FUNCTION_BLOCK FB_StepperHoming EXTENDS FB_StateMachine IMPLEMENTS  I_StateMachine
VAR_INPUT
	bStart : BOOL;	
	
	stParentsAxis : REFERENCE TO ST_StepperAxis;
	
END_VAR
VAR_OUTPUT
END_VAR
VAR
	eInnerState : E_StepperHomingStates;
	bCompleted : BOOL;
	dtTimeCompleted: DATE_AND_TIME;
	
	bEnabledBeforeHoming : BOOL;
	bOutsideHome AT %I* : BOOL;
	fRelativePosition 		: LREAL;
	fAbsolutePosition		: LREAL;
	
	stAxisRef : REFERENCE TO AXIS_REF;
	fbPower : MC_Power;
	fbReset :MC_Reset;
	fbHalt : MC_Halt;
	fbJog : MC_JOG;
	fbHome : MC_Home;
	bOutwardsForward	: REFERENCE TO BOOL;
	bOutwardsBackwards	: REFERENCE TO BOOL;
	bInwardsForward		: REFERENCE TO BOOL;
	bInwardsBackwards	: REFERENCE TO BOOL;
	fHomePosition		: REFERENCE TO LREAL;
	bForceHoming : REFERENCE TO BOOL;
	nPLC_Cycles	: INT;
END_VAR

OuterLopSM();

PROPERTY Angle : LREAL
GET
Angle := stAxisRef.NcToPlc.ActPos;
END_GET
END_PROPERTY

METHOD Disable : BOOL
bBusy := TRUE;
fbPower(Axis:=stAxisRef,Enable:=FALSE);

IF fbPower.Status = FALSE THEN
	Disable := TRUE;
ELSIF fbPower.Error THEN
	fbEventHandler(nBeckhoffID:=fbPower.ErrorID);
	{warning 'TODO: trigger e-stop'}
	Disable := TRUE;
ELSE // wait for fbPower to disable Axis 
	Disable := FALSE;
END_IF
END_METHOD

PROPERTY HomingNeeded : BOOL
GET
// TODO: Check if dtTimeCompleted is too old. If so set HomingNeeded := TRUE
IF bForceHoming THEN
	HomingNeeded := TRUE;
ELSE
	HomingNeeded := NOT bCompleted;
END_IF
END_GET
END_PROPERTY

METHOD InnerLoopSM : BOOL
// update all children FBs
fbPower(Axis:=stAxisRef);
fbReset(Axis:=stAxisRef);
fbJog(Axis:=stAxisRef);

CASE CyclicInnerCase(TO_STRING(eInnerState)) OF
	E_StepperHomingStates.Idle:
		IF bStart THEN
			bStart := FALSE;
			IF HomingNeeded THEN
				ChangeInnerState(E_StepperHomingStates.CheckIfEnabled);
			ELSE
				// Stay in Idle as homing is not needed
			END_IF
		END_IF

	E_StepperHomingStates.CheckIfEnabled:
		bEnabledBeforeHoming := fbPower.Status; // fbPower.Status = TRUE if stAxisRef is enabled
		ChangeInnerState(E_StepperHomingStates.ResetAxis1);
		
	E_StepperHomingStates.ResetAxis1:
		fbReset(Axis:=stAxisRef,Execute:=TRUE);
		nPLC_Cycles := 0;
		ChangeInnerState(E_StepperHomingStates.ResetAxis2);
		
	E_StepperHomingStates.ResetAxis2:
		nPLC_Cycles := nPLC_Cycles +1; // # of PLC cycles since reset was started
		IF fbReset.Done THEN
			IF bEnabledBeforeHoming THEN
				ChangeInnerState(E_StepperHomingStates.HomeSensorCheck);
			ELSE
				ChangeInnerState(E_StepperHomingStates.EnableAxis1);
			END_IF
		ELSIF fbReset.Error THEN
			fbEventHandler(nBeckhoffID:=fbReset.ErrorID);
			
			bError := TRUE;
		ELSE
			IF nPLC_Cycles > SystemConfig.nSTEPPER_MAX_CYCLES_TO_RESET THEN
				sErrorDetails := CONCAT3('fbReset.Done=FALSE after ',LINT_TO_STRING(SystemConfig.nSTEPPER_MAX_CYCLES_TO_RESET), ' PLC cycles');
				fbEventHandler(eNapID:=E_Event.TASK_FAILED,sMessage:=sErrorDetails);
		
				bError := TRUE;
			ELSE
				// wait... fbReset is still busy
			END_IF
			
		END_IF
		
	E_StepperHomingStates.EnableAxis1:
		fbPower(Axis:=stAxisRef,Enable:=TRUE, Enable_Positive := TRUE, Enable_Negative := TRUE);
		nPLC_Cycles := 0;
		ChangeInnerState(E_StepperHomingStates.EnableAxis2);
		
	E_StepperHomingStates.EnableAxis2:
		nPLC_Cycles := nPLC_Cycles +1; // # of PLC cycles since power command was started
		IF fbPower.Error THEN
			fbEventHandler(nBeckhoffID:=fbPower.ErrorID);
			bError := TRUE;
		ELSIF fbPower.Status = TRUE THEN // fbPower.Status = TRUE if stAxisRef is enabled
			sErrorDetails := CONCAT('# of Cycles to Enable Axis=',LINT_TO_STRING(nPLC_Cycles));
			fbEventHandler(eNapID:=E_Event.REQUEST_COMPLETED,sMessage:=sErrorDetails);
			
			fbReset(Axis:=stAxisRef,Execute:=FALSE); // reset FB to prepare it for next call 
			ChangeInnerState(E_StepperHomingStates.HomeSensorCheck);
		ELSE
			IF nPLC_Cycles > SystemConfig.nSTEPPER_MAX_CYCLES_TO_ENABLE THEN
				sErrorDetails := CONCAT3('fbPower.Status=FALSE after ',LINT_TO_STRING(SystemConfig.nSTEPPER_MAX_CYCLES_TO_ENABLE), ' PLC cycles');
				fbEventHandler(eNapID:=E_Event.TASK_FAILED,sMessage:=sErrorDetails);
		
				bError := TRUE;
			ELSE
				// Wait...	fbPower is still busy 		
			END_IF
		END_IF
		
	E_StepperHomingStates.HomeSensorCheck:
		fRelativePosition := Angle;			// save current uncalibrated position
		IF bOutsideHome THEN
			ChangeInnerState(E_StepperHomingStates.OutwardMotion);
		ELSE
			ChangeInnerState(E_StepperHomingStates.InwardMotion);
		END_IF
		
	E_StepperHomingStates.OutwardMotion:
		IF ABS(fRelativePosition - Angle) > (SystemConfig.fSTEPPER_MAX_INWARDS_POSITION + 2) THEN
			sErrorDetails := 'Unable to find home active zone after moving outwards more than the stepper max range of motion';
			fbEventHandler(eNapID:=E_Event.TASK_FAILED,sMessage:=sErrorDetails);
	
			bError := TRUE;
		ELSE
			fbJog(Axis:=stAxisRef, Mode:=MC_JOGMODE_CONTINOUS, JogForward:=bOutwardsForward, JogBackwards:=bOutwardsBackwards,Velocity:=SystemConfig.fSTEPPER_HOMING_FAST_SPEED);
			IF fbJog.Error THEN
				fbEventHandler(nBeckhoffID:=fbJog.ErrorID);
			
				bError := TRUE;
			ELSIF fbJog.CommandAborted THEN
				sErrorDetails := 'fbJog.CommandAborted=TRUE';
				fbEventHandler(eNapID:=E_Event.TASK_FAILED,sMessage:=sErrorDetails);
		
				bError := TRUE;
			ELSE
				IF fbJog.Done THEN
					sErrorDetails := 'fbJog.Done=TRUE unexpectedly';
					fbEventHandler(eNapID:=E_Event.TASK_WARNING,sMessage:=sErrorDetails);
				END_IF
				IF NOT bOutsideHome THEN
					fbJog(Axis:=stAxisRef, JogForward:=FALSE, JogBackwards:=FALSE); // reset jog
					fRelativePosition := Angle;	// save current uncalibrated position
					ChangeInnerState(E_StepperHomingStates.InwardMotion);
				ELSE 
					// wait
				END_IF
			END_IF
		END_IF

	E_StepperHomingStates.InwardMotion:
		IF ABS(fRelativePosition - Angle) > (SystemConfig.fSTEPPER_HOME_ZONE_WIDTH + 2) THEN
			sErrorDetails := 'Unable to find home active zone after moving inwards more than expected home active zone width';
			fbEventHandler(eNapID:=E_Event.TASK_FAILED,sMessage:=sErrorDetails);
	
			bError := TRUE;
		ELSE
			fbJog(Axis:=stAxisRef, Mode:=MC_JOGMODE_CONTINOUS, JogForward:=bInwardsForward, JogBackwards:=bInwardsBackwards,Velocity:=SystemConfig.fSTEPPER_HOMING_FAST_SPEED);
			IF fbJog.Error THEN
				fbEventHandler(nBeckhoffID:=fbJog.ErrorID);
			
				bError := TRUE;
			ELSIF fbJog.CommandAborted THEN
				sErrorDetails := 'fbJog.CommandAborted=TRUE';
				fbEventHandler(eNapID:=E_Event.TASK_FAILED,sMessage:=sErrorDetails);
		
				bError := TRUE;
			ELSE
				IF fbJog.Done THEN
					sErrorDetails := 'fbJog.Done=TRUE unexpectedly';
					fbEventHandler(eNapID:=E_Event.TASK_WARNING,sMessage:=sErrorDetails);
				END_IF
				IF bOutsideHome THEN
					fbJog(Axis:=stAxisRef, JogForward:=FALSE, JogBackwards:=FALSE); // reset jog
					fRelativePosition := Angle;	// save current uncalibrated position
					ChangeInnerState(E_StepperHomingStates.OutwardCreep);
				ELSE 
					// wait
				END_IF
			END_IF
		END_IF

		
	E_StepperHomingStates.OutwardCreep:
		IF ABS(fRelativePosition - Angle) > (SystemConfig.fSTEPPER_HOME_ZONE_WIDTH) THEN
			sErrorDetails := 'Unable to find home active zone after moving outwards more than expected home active zone width';
			fbEventHandler(eNapID:=E_Event.TASK_FAILED,sMessage:=sErrorDetails);
	
			bError := TRUE;
		ELSE
			IF bOutsideHome THEN
				fbJog(Axis:=stAxisRef, Mode:=MC_JOGMODE_CONTINOUS, JogForward:=bOutwardsForward, JogBackwards:=bOutwardsBackwards,Velocity:=SystemConfig.fSTEPPER_HOMING_SLOW_SPEED);
				IF fbJog.Error THEN
					fbEventHandler(nBeckhoffID:=fbJog.ErrorID);
				
					bError := TRUE;
				ELSIF fbJog.CommandAborted THEN
					sErrorDetails := 'fbJog.CommandAborted=TRUE';
					fbEventHandler(eNapID:=E_Event.TASK_FAILED,sMessage:=sErrorDetails);
			
					bError := TRUE;
				ELSE
					IF fbJog.Done THEN
						sErrorDetails := 'fbJog.Done=TRUE unexpectedly';
						fbEventHandler(eNapID:=E_Event.TASK_WARNING,sMessage:=sErrorDetails);
					END_IF
					// wait... fbJog.busy (moving) 
				END_IF
			ELSE
				fbJog(Axis:=stAxisRef, JogForward:=FALSE, JogBackwards:=FALSE); // reset jog
				fRelativePosition := Angle;	// save current uncalibrated position
				ChangeInnerState(E_StepperHomingStates.WaitingForHalt);
			END_IF
		END_IF
		
	E_StepperHomingStates.WaitingForHalt:
		fbHalt(Axis:=stAxisRef,Execute:=TRUE);
		IF fbHalt.Done THEN
			fbHalt(Axis:=stAxisRef,Execute:=FALSE);
			ChangeInnerState(E_StepperHomingStates.GettingCurrentPos);
		ELSIF fbHalt.Error THEN
			fbEventHandler(nBeckhoffID:=fbHalt.ErrorID);
				
			bError := TRUE;
		ELSE
			// wait... fbHalt.busy
		END_IF

	E_StepperHomingStates.GettingCurrentPos:
		fAbsolutePosition := fHomePosition + (Angle - fRelativePosition);
		ChangeInnerState(E_StepperHomingStates.SettingHomePos);
	
	E_StepperHomingStates.SettingHomePos:
		fbHome(Axis:=stAxisRef, Execute:=TRUE, Position:=fAbsolutePosition, HomingMode:=MC_HomingMode.MC_Direct);
		IF fbHome.Error THEN
			fbEventHandler(nBeckhoffID:=fbHome.ErrorID);
		
			bError := TRUE;
		ELSIF fbHome.CommandAborted THEN
			sErrorDetails := 'fbHome.CommandAborted=TRUE';
			fbEventHandler(eNapID:=E_Event.TASK_FAILED,sMessage:=sErrorDetails);
	
			bError := TRUE;
		ELSIF fbHome.Done THEN
			fbHome(Axis:=stAxisRef, Execute:=FALSE); // reset homing command
			IF bEnabledBeforeHoming THEN
				ChangeInnerState(E_StepperHomingStates.WrapUp);
			ELSE
				ChangeInnerState(E_StepperHomingStates.DisableAxis);
			END_IF
		ELSE
			// wait... fbHome.busy
		END_IF
		
	E_StepperHomingStates.DisableAxis:
		fbPower(Axis:=stAxisRef,Enable:=FALSE);
		IF fbPower.Error THEN
			fbEventHandler(nBeckhoffID:=fbPower.ErrorID);
			bError := TRUE;
		ELSIF fbPower.Status = FALSE THEN // fbPower.Status = FALSE if stAxisRef is disabled
			ChangeInnerState(E_StepperHomingStates.WrapUp);
		ELSE
			// Wait...	fbPower is still busy 		
		END_IF

	
	E_StepperHomingStates.WrapUp:
		bCompleted := TRUE;
		dtTimeCompleted := DateTime.GVL_DATE_TIME;
		ChangeInnerState(E_StepperHomingStates.Idle);
END_CASE
END_METHOD

METHOD Reset : BOOL
// reset variables specific to this FB 
bCompleted := FALSE;
dtTimeCompleted := DATE_AND_TIME#1970-1-1-0:0:0;

// Reactivate children FBs
//none
END_METHOD

METHOD Setup : BOOL
eStateMachineSourceID := eStateSourceID;
stAxisRef REF= stParentsAxis.stAxisRef;

bOutwardsForward 	REF= stParentsAxis.bOutwardsForward;
bOutwardsBackwards	REF= stParentsAxis.bOutwardsBackwards;
bInwardsForward		REF= stParentsAxis.bInwardsForward;
bInwardsBackwards	REF= stParentsAxis.bInwardsBackwards;
fHomePosition		REF= stParentsAxis.fHomePosition;
bForceHoming REF= stParentsAxis.bForceHoming;

SetInnerEnumeration(nStateEnum:=THIS^.eInnerState);
END_METHOD

PROPERTY TimeCompleted : DATE_AND_TIME
GET
TimeCompleted := dtTimeCompleted;
END_GET
END_PROPERTY

END_FUNCTION_BLOCK

(* stored: Version 1.1.0.1, ProductVersion 3.1.4024.12
   POU FB_StepperHoming: Id {02f8ef0c-5a00-4080-a395-cb849d80913d}, SpecialFunc None
   Folder Properties: Id {16e96894-613b-4510-b160-c7745d2583f5}
   Property Angle: Id {d5e9e495-261b-48a4-a146-d0b6127ddca7}
   Get Get: Id {3ce02f1e-fa30-4779-86c3-afa2141de322}
   Method Disable: Id {2cb3ba08-48bc-4ada-b68b-4bc909bee3d1}
   Property HomingNeeded: Id {b520ae64-639c-45df-8d50-027d7c3a6b31}
   Get Get: Id {c8d57e3f-f04f-464a-8306-fceb94c76e94}
   Method InnerLoopSM: Id {6520a2ec-f048-42e4-86c6-b710b0c82fde}
   Method Reset: Id {f0bd47d6-c200-481f-868a-da6daf0066cc}
   Method Setup: Id {38ac2a80-93ba-4a8f-b6b0-8eb833401930}
   Property TimeCompleted: Id {09f49961-ab82-4f90-9aa9-2db523e21ec7}
   Get Get: Id {4445d525-ba0b-4652-81d7-5602accba4d9} *)
